// TIA Portal V15.1 export
// export: Created 2024-05-17T05:38:54.0662979Z, ExportSetting WithDefaults, DisplayName Totally Integrated Automation Portal, DisplayVersion V15.1 Update 5, DisplayName TIA Portal Openness, DisplayVersion V15.1 Update 5, DisplayName SINAMICS Startdrive Advanced, DisplayVersion V15.1, DisplayName G130, G150, S120, S150, SINAMICS MV, S210, DisplayVersion V15.1, DisplayName G110M, G120, G120C, G120D, G120P, DisplayVersion V15.1, DisplayName STEP 7 Professional, DisplayVersion V15.1 Update 5, DisplayName STEP 7 Safety, DisplayVersion V15.1, DisplayName WinCC Professional, DisplayVersion V15.1 Update 5, DisplayName SIMATIC Visualization Architect, DisplayVersion V15.1
FUNCTION_BLOCK "LVIDSTrack"   // FB1205, FBD
TITLE = LVIDS Tracking
{ S7_Optimized_Access := 'TRUE' }
VERSION : 0.1
// stored: AutoNumber false, IsIECCheckEnabled false, IsRetainMemResEnabled false, MemoryReserve 100, SetENOAutomatically False, UDAEnableTagReadback false
   VAR_INPUT
      I_DataModeManEn { ExternalAccessible := 'False'; ExternalVisible := 'False'; ExternalWritable := 'False'} : Bool;   // Data mode manual enabled
      I_OutOfUse { ExternalAccessible := 'False'; ExternalVisible := 'False'; ExternalWritable := 'False'} : Bool;   // Out of use
      I_TagID { ExternalAccessible := 'False'; ExternalVisible := 'False'; ExternalWritable := 'False'} : DInt;   // Tag identification for tracking
      I_BodyID { ExternalAccessible := 'False'; ExternalVisible := 'False'; ExternalWritable := 'False'} : DInt;   // Body identification for tracking
      I_CarrierID { ExternalAccessible := 'False'; ExternalVisible := 'False'; ExternalWritable := 'False'} : DInt;   // Carrier identification for tracking
      I_MixNbr { ExternalAccessible := 'False'; ExternalVisible := 'False'; ExternalWritable := 'False'} : DInt;   // Mixnumber for tracking
      I_BodyType1 { ExternalAccessible := 'False'; ExternalVisible := 'False'; ExternalWritable := 'False'} : DInt;   // Bodytype1 for tracking
      I_PopID { ExternalAccessible := 'False'; ExternalVisible := 'False'; ExternalWritable := 'False'} : UDInt;   // Spare Data / PopID
      I_PopIDSuffix { ExternalAccessible := 'False'; ExternalVisible := 'False'; ExternalWritable := 'False'} : Char;   // PopID suffix
      I_PopType { ExternalAccessible := 'False'; ExternalVisible := 'False'; ExternalWritable := 'False'} : UDInt;   // Pop identifier
      I_Start { ExternalAccessible := 'False'; ExternalVisible := 'False'; ExternalWritable := 'False'} : Bool;   // Start function / Start track
   END_VAR
   VAR_OUTPUT
      O_Ok { ExternalAccessible := 'False'; ExternalVisible := 'False'; ExternalWritable := 'False'} : Bool;   // Function finished / OK
      O_Nok { ExternalAccessible := 'False'; ExternalVisible := 'False'; ExternalWritable := 'False'} : Bool;   // NOK
      O_Busy { ExternalAccessible := 'False'; ExternalVisible := 'False'; ExternalWritable := 'False'} : Bool;   // Busy
      O_Status { ExternalAccessible := 'False'; ExternalVisible := 'False'; ExternalWritable := 'False'} : Int;   // Status ( < 0 : Fault ; 0 : No status; 1 : Success ; > 1 : Busy)
      O_Alarm { ExternalAccessible := 'False'; ExternalVisible := 'False'; ExternalWritable := 'False'} : Bool;   // Alarm
   END_VAR
   VAR_IN_OUT
      IO_VIDS : "VIDS";   // VIDS - internal record
      IO_Alarm : "Alarm";   // Alarm
      H_Track : "H_LVIDSTrack";   // Animation
      H_HMI : "H_HMI";   // Animation
   END_VAR
   VAR
      BtnManTrack { ExternalAccessible := 'False'; ExternalVisible := 'False'; ExternalWritable := 'False'} : Bool;
      BtnManForce { ExternalAccessible := 'False'; ExternalVisible := 'False'; ExternalWritable := 'False'} : Bool;
      BtnManOK { ExternalAccessible := 'False'; ExternalVisible := 'False'; ExternalWritable := 'False'} : Bool;
      BlockAutoStart { ExternalAccessible := 'False'; ExternalVisible := 'False'; ExternalWritable := 'False'} : Bool;
      RSAutoBlock { ExternalAccessible := 'False'; ExternalVisible := 'False'; ExternalWritable := 'False'} : Bool;
      TagIDMem { ExternalAccessible := 'False'; ExternalVisible := 'False'; ExternalWritable := 'False'} : DWord;
      BodyNbrMem { ExternalAccessible := 'False'; ExternalVisible := 'False'; ExternalWritable := 'False'} : DWord;
      MixNbrMem { ExternalAccessible := 'False'; ExternalVisible := 'False'; ExternalWritable := 'False'} : DWord;
      CarrierIDMem { ExternalAccessible := 'False'; ExternalVisible := 'False'; ExternalWritable := 'False'} : DWord;
      BodyType1Mem { ExternalAccessible := 'False'; ExternalVisible := 'False'; ExternalWritable := 'False'} : DWord;
      PopIDMem { ExternalAccessible := 'False'; ExternalVisible := 'False'; ExternalWritable := 'False'} : DWord;
      PopIDSuffixMem { ExternalAccessible := 'False'; ExternalVisible := 'False'; ExternalWritable := 'False'} : Char;
      PopTypeMem { ExternalAccessible := 'False'; ExternalVisible := 'False'; ExternalWritable := 'False'} : DWord;
      StartEdg { ExternalAccessible := 'False'; ExternalVisible := 'False'; ExternalWritable := 'False'} : Bool;   // Edge of start tracking
      StartPls { ExternalAccessible := 'False'; ExternalVisible := 'False'; ExternalWritable := 'False'} : Bool;
      StartTrackEdge2 { ExternalAccessible := 'False'; ExternalVisible := 'False'; ExternalWritable := 'False'} : Bool;   // Edge of start tracking
      StartCmdMem { ExternalAccessible := 'False'; ExternalVisible := 'False'; ExternalWritable := 'False'} : Bool;   // Memory of start command
      FinishPls { ExternalAccessible := 'False'; ExternalVisible := 'False'; ExternalWritable := 'False'} : Bool;   // Pulse of finish tracking
      FinishEdge { ExternalAccessible := 'False'; ExternalVisible := 'False'; ExternalWritable := 'False'} : Bool;   // Edge of finish tracking
      Status { ExternalAccessible := 'False'; ExternalVisible := 'False'; ExternalWritable := 'False'} : Int;   // Status
      Alarm { ExternalAccessible := 'False'; ExternalVisible := 'False'; ExternalWritable := 'False'} : Bool;
      Ok { ExternalAccessible := 'False'; ExternalVisible := 'False'; ExternalWritable := 'False'} : Bool;
      Nok { ExternalAccessible := 'False'; ExternalVisible := 'False'; ExternalWritable := 'False'} : Bool;
      BtnManConfirmVisible { ExternalAccessible := 'False'; ExternalVisible := 'False'; ExternalWritable := 'False'} : Word;
      BtnManConfirmGreen { ExternalAccessible := 'False'; ExternalVisible := 'False'; ExternalWritable := 'False'} : Word;
      BtnManForceVisible { ExternalAccessible := 'False'; ExternalVisible := 'False'; ExternalWritable := 'False'} : Word;
      BtnManForceGreen { ExternalAccessible := 'False'; ExternalVisible := 'False'; ExternalWritable := 'False'} : Word;
   END_VAR
   VAR_TEMP
      TempNotUsedBool : Bool;
   END_VAR
   VAR CONSTANT
      CMD_TRACK : DWord := 4001;
      OFF : Word := 2#0000000000000000;
      ENABLE : Word := 2#0000000000000001;
      VISIBLE : Word := 2#0000000000000010;
      COLOUR_GREY : Word := 2#0000000000010000;
      COLOUR_WHITE : Word := 2#0000000000100000;
      COLOUR_GREEN : Word := 2#0000000001000000;
      COLOUR_RED : Word := 2#0000000010000000;
      COLOUR_BLUE_FLASH : Word := 2#0000000100000000;
   END_VAR
   VAR_TEMP   // added for the SCL form of the ladder/FBD networks
      _w1 : Bool;
   END_VAR
BEGIN

REGION Network 1: **** 4.4 - Machine status - Input from HMI - Buttons
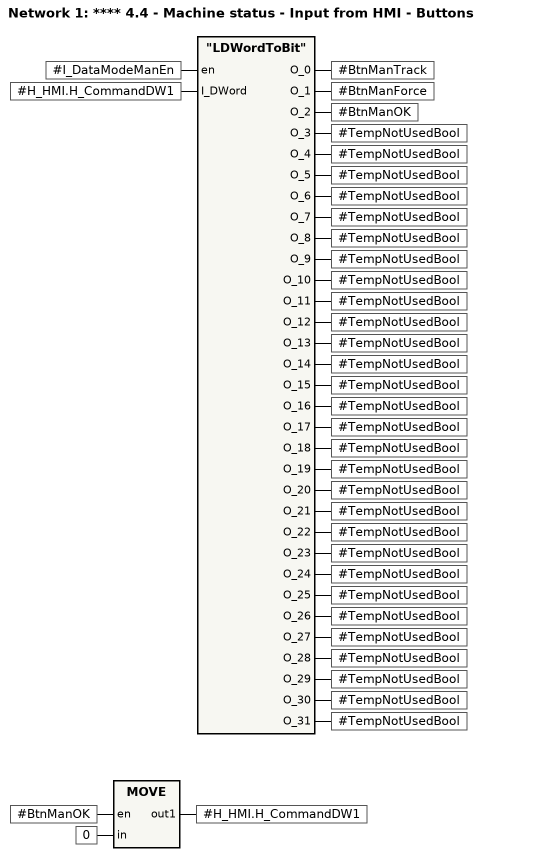
   IF #I_DataModeManEn THEN
       "LDWordToBit"(I_DWord := #H_HMI.H_CommandDW1,
                     O_0 => #BtnManTrack,
                     O_1 => #BtnManForce,
                     O_2 => #BtnManOK,
                     O_3 => #TempNotUsedBool,
                     O_4 => #TempNotUsedBool,
                     O_5 => #TempNotUsedBool,
                     O_6 => #TempNotUsedBool,
                     O_7 => #TempNotUsedBool,
                     O_8 => #TempNotUsedBool,
                     O_9 => #TempNotUsedBool,
                     O_10 => #TempNotUsedBool,
                     O_11 => #TempNotUsedBool,
                     O_12 => #TempNotUsedBool,
                     O_13 => #TempNotUsedBool,
                     O_14 => #TempNotUsedBool,
                     O_15 => #TempNotUsedBool,
                     O_16 => #TempNotUsedBool,
                     O_17 => #TempNotUsedBool,
                     O_18 => #TempNotUsedBool,
                     O_19 => #TempNotUsedBool,
                     O_20 => #TempNotUsedBool,
                     O_21 => #TempNotUsedBool,
                     O_22 => #TempNotUsedBool,
                     O_23 => #TempNotUsedBool,
                     O_24 => #TempNotUsedBool,
                     O_25 => #TempNotUsedBool,
                     O_26 => #TempNotUsedBool,
                     O_27 => #TempNotUsedBool,
                     O_28 => #TempNotUsedBool,
                     O_29 => #TempNotUsedBool,
                     O_30 => #TempNotUsedBool,
                     O_31 => #TempNotUsedBool);
   END_IF;
   IF #BtnManOK THEN #H_HMI.H_CommandDW1 := 0; END_IF;
END_REGION

REGION Network 2: *** 4.4 - Machine status - Calculated *** / **** 4.4 - Machine status - Calculated *** Begin request
   // Start request memory
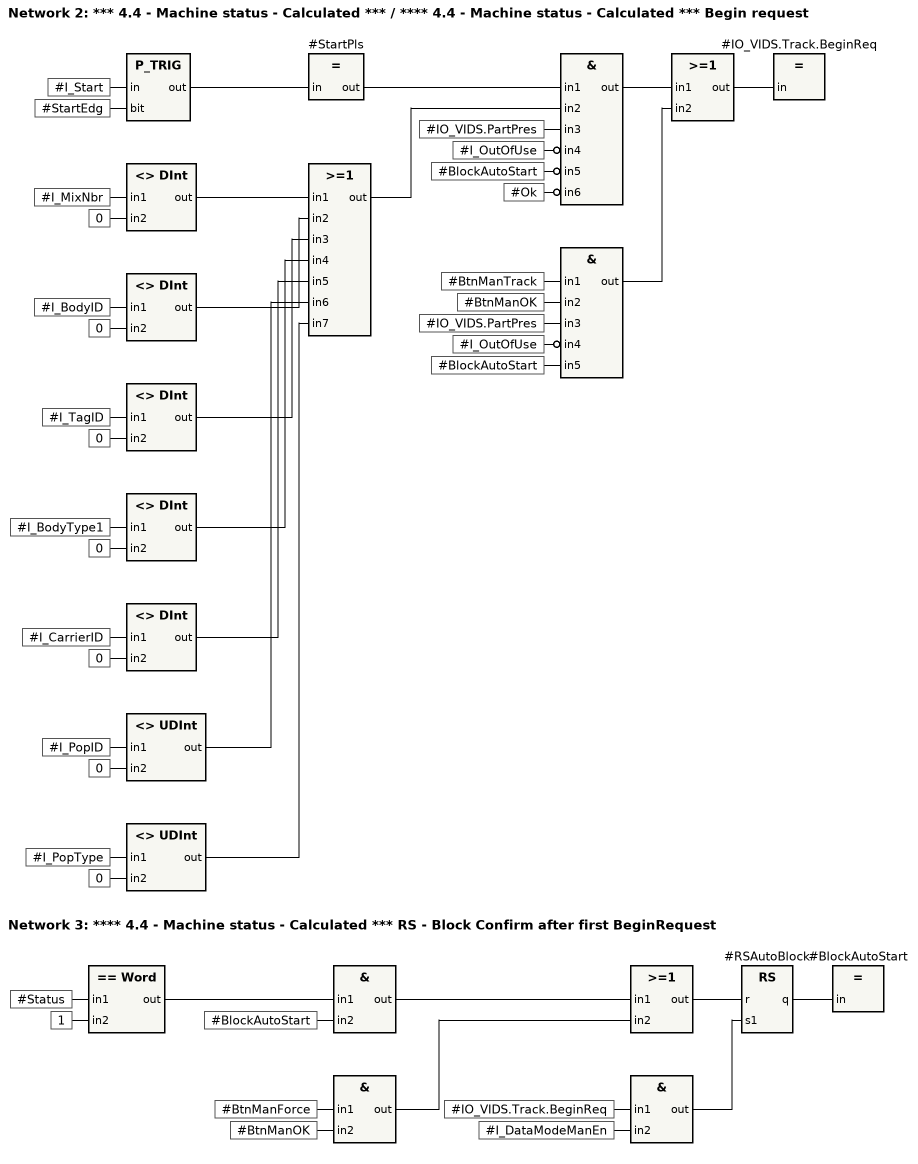
   #_w1 := #I_Start AND NOT #StartEdg;   // rising edge
   #StartEdg := #I_Start;
   #StartPls := #_w1;
   #IO_VIDS.Track.BeginReq := (#_w1 AND ((#I_MixNbr <> 0) OR (#I_BodyID <> 0) OR (#I_TagID <> 0) OR (#I_BodyType1 <> 0) OR (#I_CarrierID <> 0) OR (#I_PopID <> 0) OR (#I_PopType <> 0)) AND #IO_VIDS.PartPres AND NOT #I_OutOfUse AND NOT #BlockAutoStart AND NOT #Ok) OR (#BtnManTrack AND #BtnManOK AND #IO_VIDS.PartPres AND NOT #I_OutOfUse AND #BlockAutoStart);
END_REGION

REGION Network 3: **** 4.4 - Machine status - Calculated *** RS - Block Confirm after first BeginRequest
   IF ((#Status = 1) AND #BlockAutoStart) OR (#BtnManForce AND #BtnManOK) THEN
       #RSAutoBlock := FALSE;   // RS flip-flop
   END_IF;
   IF #IO_VIDS.Track.BeginReq AND #I_DataModeManEn THEN #RSAutoBlock := TRUE; END_IF;
   #BlockAutoStart := #RSAutoBlock;
END_REGION

REGION Network 4: **** 4.4 - Machine status - Calculated *** Memorize parameters
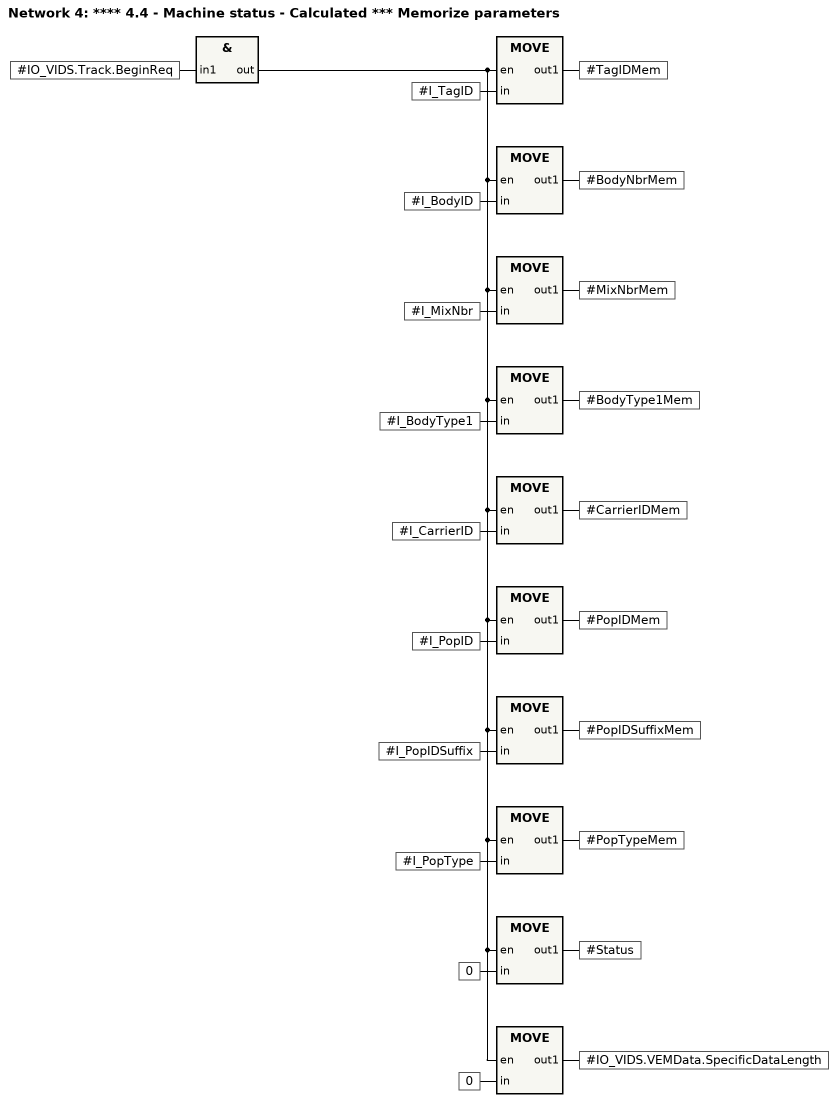
   IF #IO_VIDS.Track.BeginReq THEN
       #TagIDMem := #I_TagID;
       #BodyNbrMem := #I_BodyID;
       #MixNbrMem := #I_MixNbr;
       #BodyType1Mem := #I_BodyType1;
       #CarrierIDMem := #I_CarrierID;
       #PopIDMem := #I_PopID;
       #PopIDSuffixMem := #I_PopIDSuffix;
       #PopTypeMem := #I_PopType;
       #Status := 0;
       #IO_VIDS.VEMData.SpecificDataLength := 0;
   END_IF;
END_REGION

REGION Network 5: *** 4.4 - Machine status - Calculated *** / **** 4.4 - Machine status - Calculated *** Ok to begin
   // Data mode auto - Begin pulse
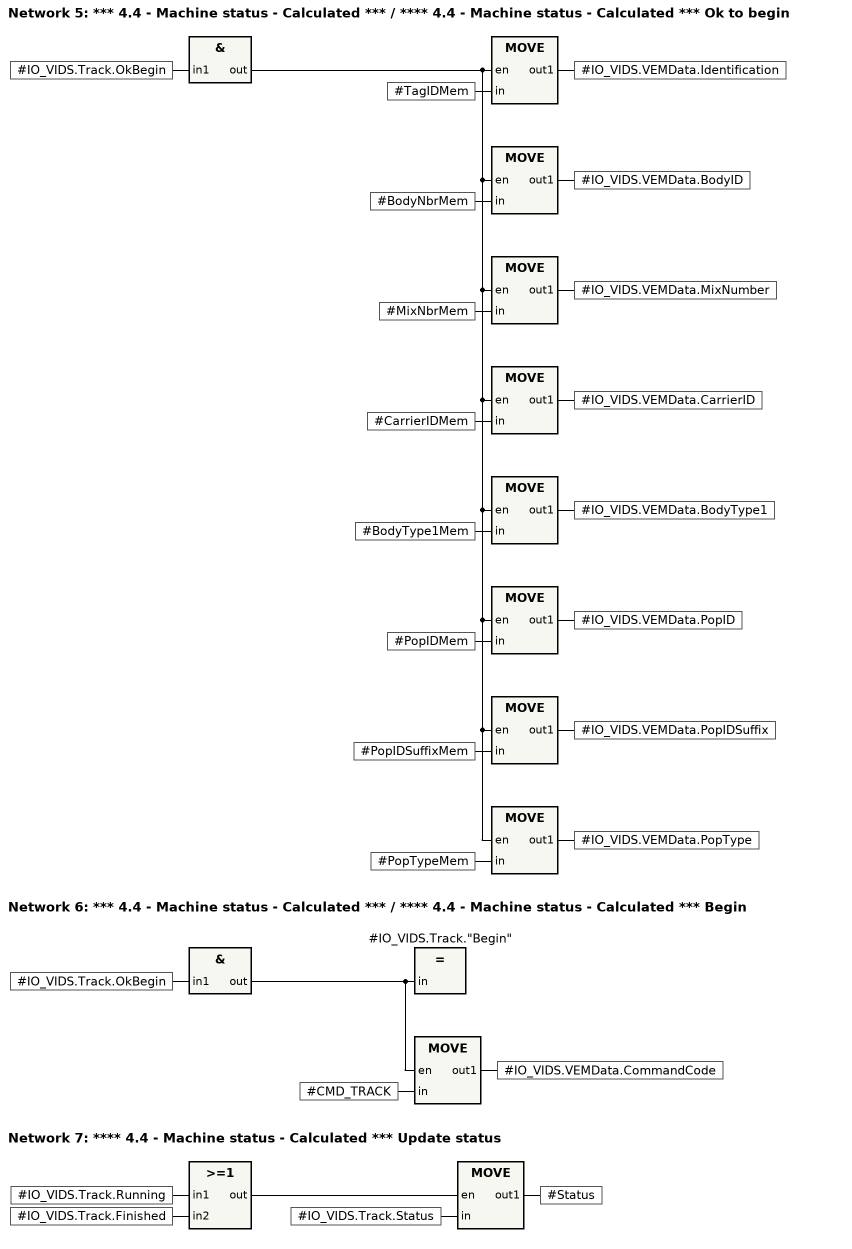
   IF #IO_VIDS.Track.OkBegin THEN
       #IO_VIDS.VEMData.Identification := #TagIDMem;
       #IO_VIDS.VEMData.BodyID := #BodyNbrMem;
       #IO_VIDS.VEMData.MixNumber := #MixNbrMem;
       #IO_VIDS.VEMData.CarrierID := #CarrierIDMem;
       #IO_VIDS.VEMData.BodyType1 := #BodyType1Mem;
       #IO_VIDS.VEMData.PopID := #PopIDMem;
       #IO_VIDS.VEMData.PopIDSuffix := #PopIDSuffixMem;
       #IO_VIDS.VEMData.PopType := #PopTypeMem;
   END_IF;
END_REGION

REGION Network 6: *** 4.4 - Machine status - Calculated *** / **** 4.4 - Machine status - Calculated *** Begin
   // Data mode auto - Begin pulse
   #IO_VIDS.Track."Begin" := #IO_VIDS.Track.OkBegin;
   IF #IO_VIDS.Track.OkBegin THEN #IO_VIDS.VEMData.CommandCode := #CMD_TRACK; END_IF;
END_REGION

REGION Network 7: **** 4.4 - Machine status - Calculated *** Update status
   IF #IO_VIDS.Track.Running OR #IO_VIDS.Track.Finished THEN #Status := #IO_VIDS.Track.Status; END_IF;
END_REGION

REGION Network 8: *** 8 - Outputs *** / **** 4.4 - Machine status - Calculated *** Finished, OK
   // Feedback to process - Tracking finished
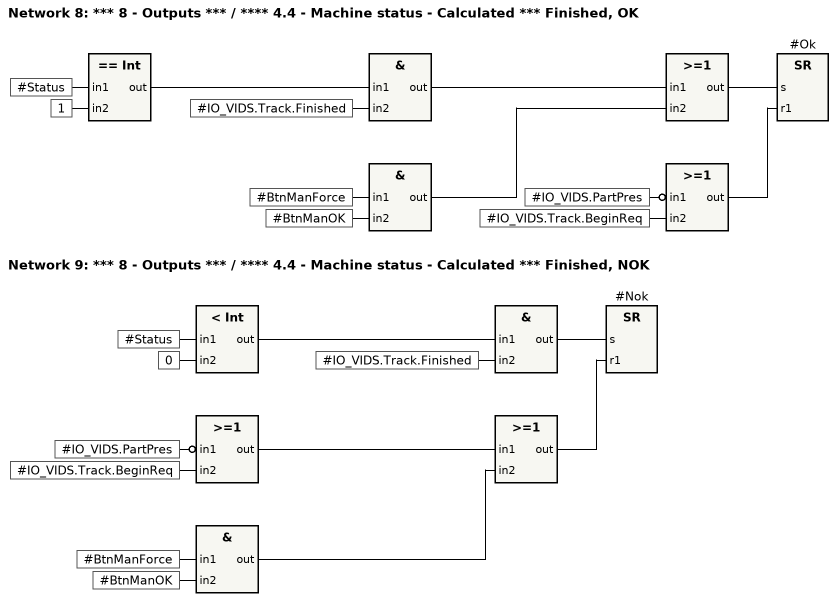
   IF ((#Status = 1) AND #IO_VIDS.Track.Finished) OR (#BtnManForce AND #BtnManOK) THEN
       #Ok := TRUE;   // SR flip-flop
   END_IF;
   IF NOT #IO_VIDS.PartPres OR #IO_VIDS.Track.BeginReq THEN #Ok := FALSE; END_IF;
END_REGION

REGION Network 9: *** 8 - Outputs *** / **** 4.4 - Machine status - Calculated *** Finished, NOK
   // Feedback to process - Tracking finished
   IF (#Status < 0) AND #IO_VIDS.Track.Finished THEN
       #Nok := TRUE;   // SR flip-flop
   END_IF;
   IF NOT #IO_VIDS.PartPres OR #IO_VIDS.Track.BeginReq OR (#BtnManForce AND #BtnManOK) THEN
       #Nok := FALSE;
   END_IF;
END_REGION

REGION Network 10: **** 4.6 - Machine status - Indication *** To HMI - Reset HMI parameters
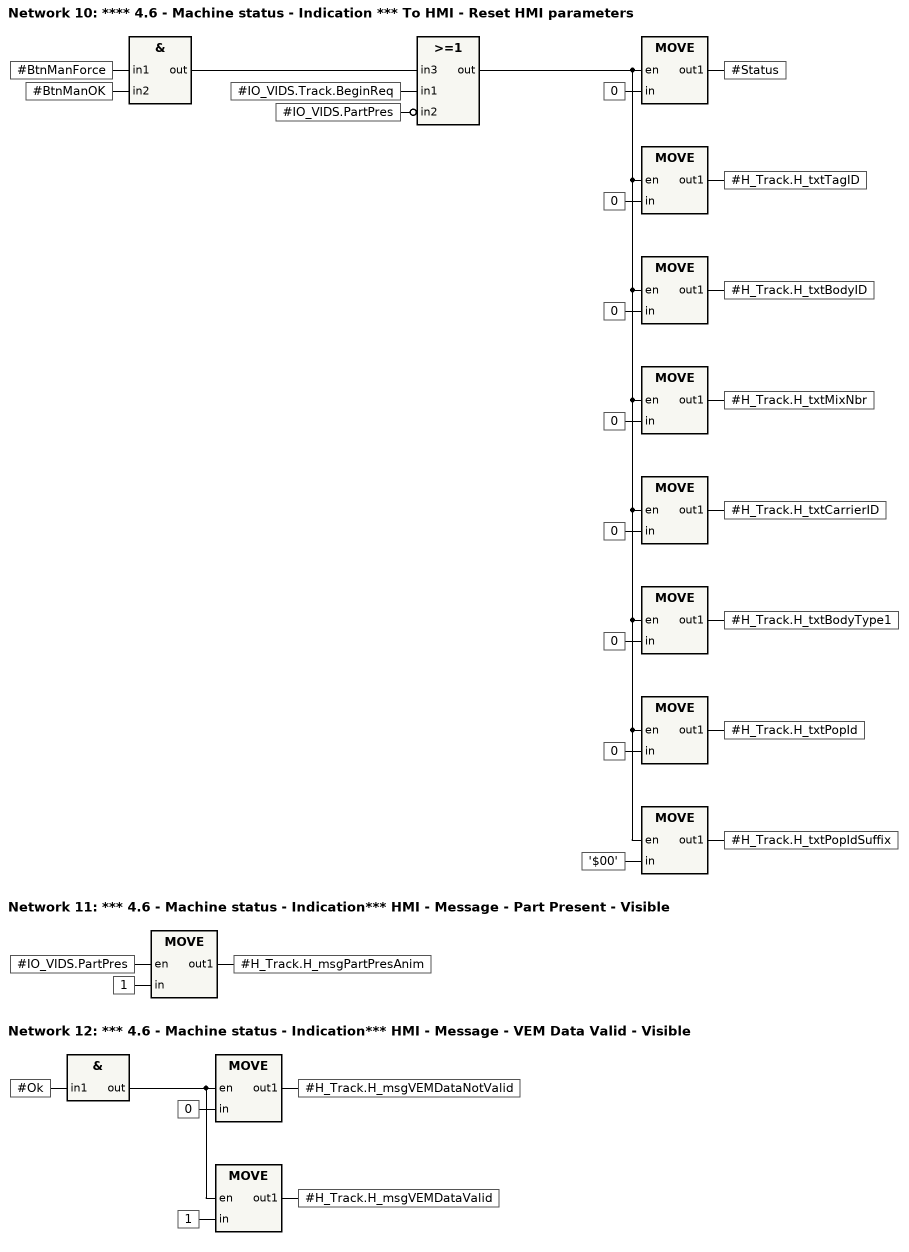
   IF (#BtnManForce AND #BtnManOK) OR #IO_VIDS.Track.BeginReq OR NOT #IO_VIDS.PartPres THEN
       #Status := 0;
       #H_Track.H_txtTagID := 0;
       #H_Track.H_txtBodyID := 0;
       #H_Track.H_txtMixNbr := 0;
       #H_Track.H_txtCarrierID := 0;
       #H_Track.H_txtBodyType1 := 0;
       #H_Track.H_txtPopId := 0;
       #H_Track.H_txtPopIdSuffix := '$00';
   END_IF;
END_REGION

REGION Network 11: *** 4.6 - Machine status - Indication*** HMI - Message - Part Present - Visible
   IF #IO_VIDS.PartPres THEN #H_Track.H_msgPartPresAnim := 1; END_IF;
END_REGION

REGION Network 12: *** 4.6 - Machine status - Indication*** HMI - Message - VEM Data Valid - Visible
   IF #Ok THEN
       #H_Track.H_msgVEMDataNotValid := 0;
       #H_Track.H_msgVEMDataValid := 1;
   END_IF;
END_REGION

REGION Network 13: *** 4.6 - Machine status - Indication*** HMI - Message - VEM Data Not Valid - Visible
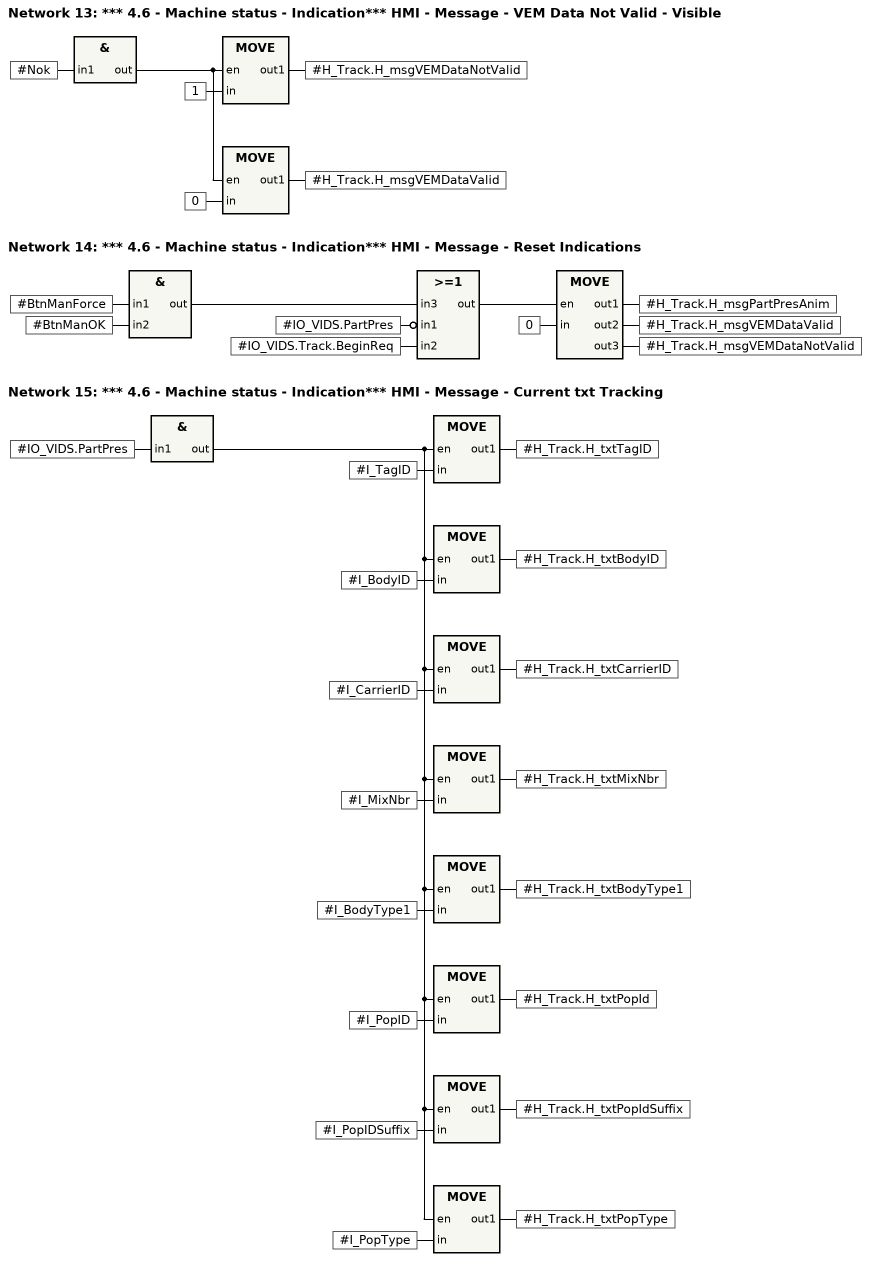
   IF #Nok THEN
       #H_Track.H_msgVEMDataNotValid := 1;
       #H_Track.H_msgVEMDataValid := 0;
   END_IF;
END_REGION

REGION Network 14: *** 4.6 - Machine status - Indication*** HMI - Message - Reset Indications
   IF (#BtnManForce AND #BtnManOK) OR NOT #IO_VIDS.PartPres OR #IO_VIDS.Track.BeginReq THEN
       #H_Track.H_msgPartPresAnim := 0;
       #H_Track.H_msgVEMDataValid := 0;
       #H_Track.H_msgVEMDataNotValid := 0;
   END_IF;
END_REGION

REGION Network 15: *** 4.6 - Machine status - Indication*** HMI - Message - Current txt Tracking
   IF #IO_VIDS.PartPres THEN
       #H_Track.H_txtTagID := #I_TagID;
       #H_Track.H_txtBodyID := #I_BodyID;
       #H_Track.H_txtCarrierID := #I_CarrierID;
       #H_Track.H_txtMixNbr := #I_MixNbr;
       #H_Track.H_txtBodyType1 := #I_BodyType1;
       #H_Track.H_txtPopId := #I_PopID;
       #H_Track.H_txtPopIdSuffix := #I_PopIDSuffix;
       #H_Track.H_txtPopType := #I_PopType;
   END_IF;
END_REGION

REGION Network 16: *** 4.6 - Machine status - Indication*** HMI - Message - Current txt Tracking Reset
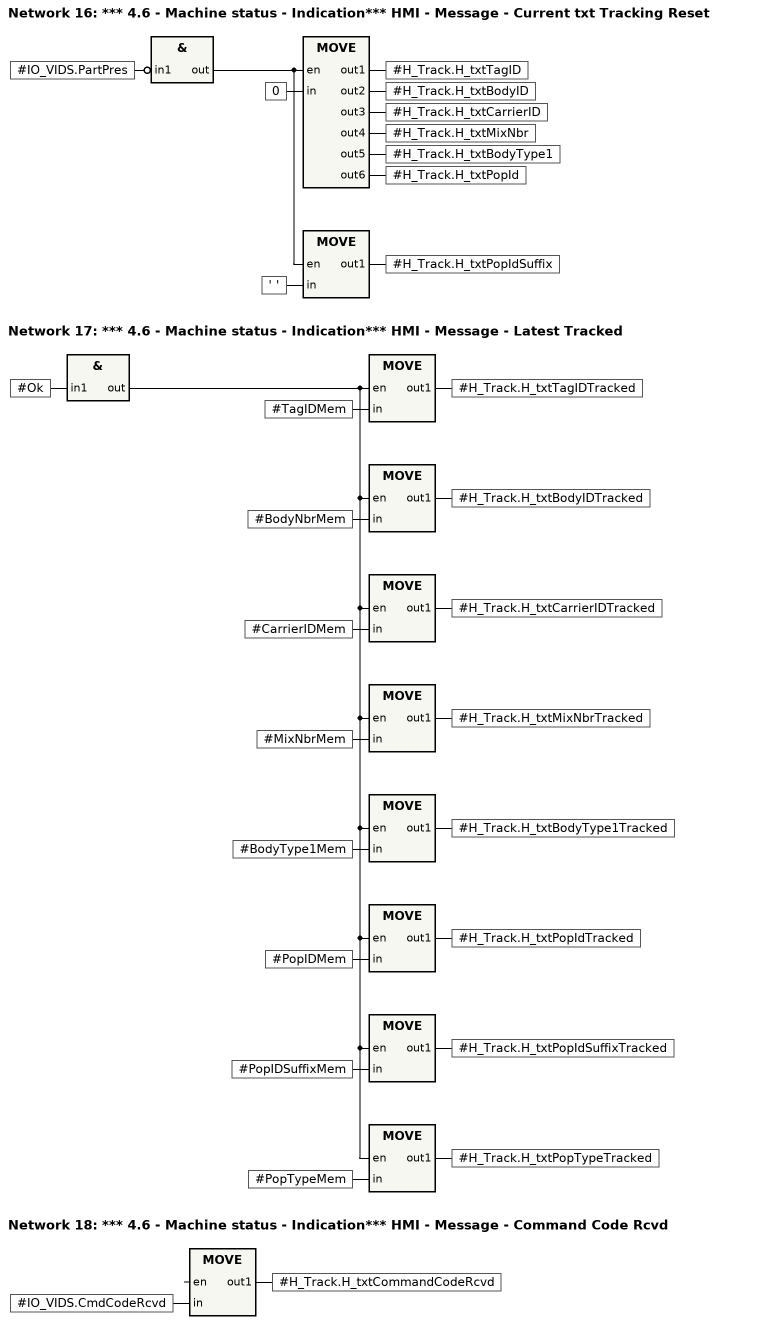
   IF NOT #IO_VIDS.PartPres THEN
       #H_Track.H_txtTagID := 0;
       #H_Track.H_txtBodyID := 0;
       #H_Track.H_txtCarrierID := 0;
       #H_Track.H_txtMixNbr := 0;
       #H_Track.H_txtBodyType1 := 0;
       #H_Track.H_txtPopId := 0;
       #H_Track.H_txtPopIdSuffix := ' ';
   END_IF;
END_REGION

REGION Network 17: *** 4.6 - Machine status - Indication*** HMI - Message - Latest Tracked
   IF #Ok THEN
       #H_Track.H_txtTagIDTracked := #TagIDMem;
       #H_Track.H_txtBodyIDTracked := #BodyNbrMem;
       #H_Track.H_txtCarrierIDTracked := #CarrierIDMem;
       #H_Track.H_txtMixNbrTracked := #MixNbrMem;
       #H_Track.H_txtBodyType1Tracked := #BodyType1Mem;
       #H_Track.H_txtPopIdTracked := #PopIDMem;
       #H_Track.H_txtPopIdSuffixTracked := #PopIDSuffixMem;
       #H_Track.H_txtPopTypeTracked := #PopTypeMem;
   END_IF;
END_REGION

REGION Network 18: *** 4.6 - Machine status - Indication*** HMI - Message - Command Code Rcvd
   #H_Track.H_txtCommandCodeRcvd := #IO_VIDS.CmdCodeRcvd;
END_REGION

REGION Network 19: *** 4.6 - Machine status - Indication*** HMI - Message - Command Code Sent
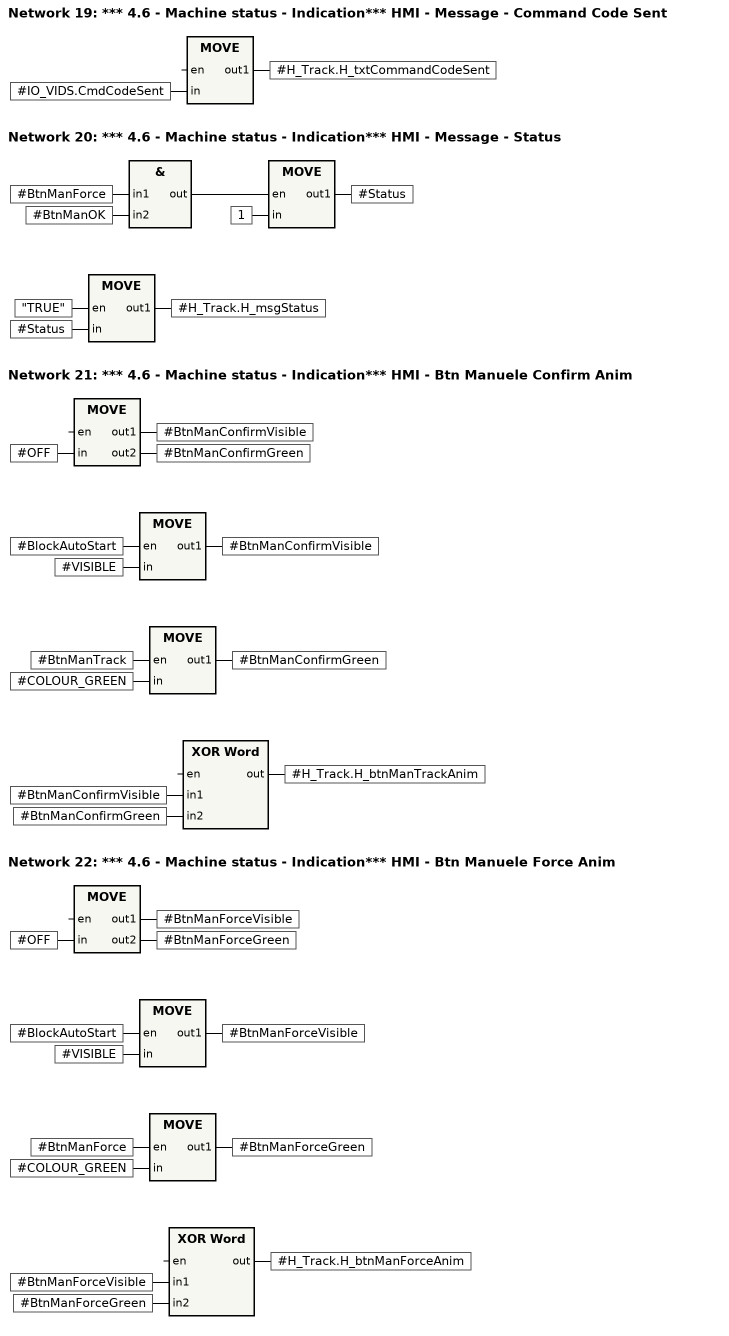
   #H_Track.H_txtCommandCodeSent := #IO_VIDS.CmdCodeSent;
END_REGION

REGION Network 20: *** 4.6 - Machine status - Indication*** HMI - Message - Status
   IF #BtnManForce AND #BtnManOK THEN #Status := 1; END_IF;
   IF "TRUE" THEN #H_Track.H_msgStatus := #Status; END_IF;
END_REGION

REGION Network 21: *** 4.6 - Machine status - Indication*** HMI - Btn Manuele Confirm Anim
   #BtnManConfirmVisible := #OFF;
   #BtnManConfirmGreen := #OFF;
   IF #BlockAutoStart THEN #BtnManConfirmVisible := #VISIBLE; END_IF;
   IF #BtnManTrack THEN #BtnManConfirmGreen := #COLOUR_GREEN; END_IF;
   #H_Track.H_btnManTrackAnim := #BtnManConfirmVisible XOR #BtnManConfirmGreen;
END_REGION

REGION Network 22: *** 4.6 - Machine status - Indication*** HMI - Btn Manuele Force Anim
   #BtnManForceVisible := #OFF;
   #BtnManForceGreen := #OFF;
   IF #BlockAutoStart THEN #BtnManForceVisible := #VISIBLE; END_IF;
   IF #BtnManForce THEN #BtnManForceGreen := #COLOUR_GREEN; END_IF;
   #H_Track.H_btnManForceAnim := #BtnManForceVisible XOR #BtnManForceGreen;
END_REGION

REGION Network 23: *** 4.6 - Machine status - Indication*** HMI - Btn Manuele Confirm Anim
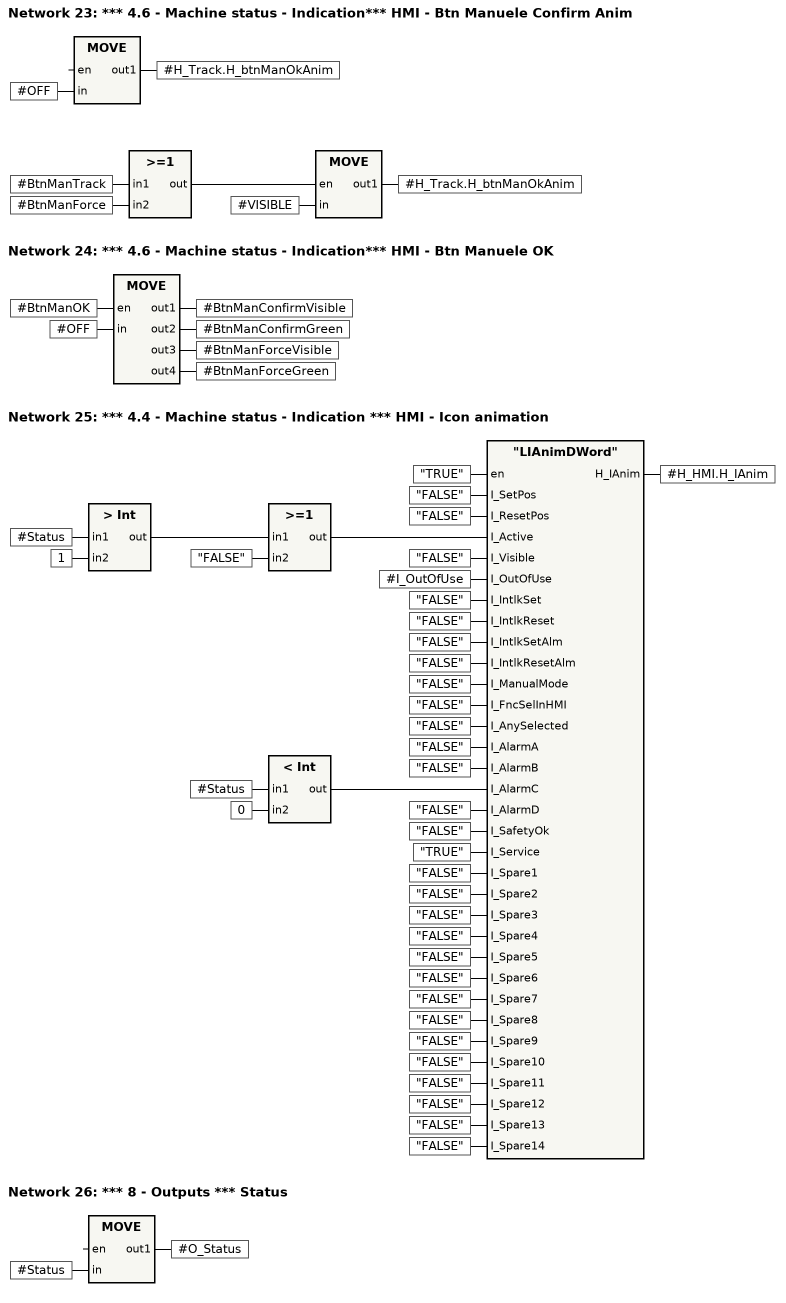
   #H_Track.H_btnManOkAnim := #OFF;
   IF #BtnManTrack OR #BtnManForce THEN #H_Track.H_btnManOkAnim := #VISIBLE; END_IF;
END_REGION

REGION Network 24: *** 4.6 - Machine status - Indication*** HMI - Btn Manuele OK
   IF #BtnManOK THEN
       #BtnManConfirmVisible := #OFF;
       #BtnManConfirmGreen := #OFF;
       #BtnManForceVisible := #OFF;
       #BtnManForceGreen := #OFF;
   END_IF;
END_REGION

REGION Network 25: *** 4.4 - Machine status - Indication *** HMI - Icon animation
   IF "TRUE" THEN
       "LIAnimDWord"(I_SetPos := "FALSE",
                     I_ResetPos := "FALSE",
                     I_Active := (#Status > 1) OR "FALSE",
                     I_Visible := "FALSE",
                     I_OutOfUse := #I_OutOfUse,
                     I_IntlkSet := "FALSE",
                     I_IntlkReset := "FALSE",
                     I_IntlkSetAlm := "FALSE",
                     I_IntlkResetAlm := "FALSE",
                     I_ManualMode := "FALSE",
                     I_FncSelInHMI := "FALSE",
                     I_AnySelected := "FALSE",
                     I_AlarmA := "FALSE",
                     I_AlarmB := "FALSE",
                     I_AlarmC := #Status < 0,
                     I_AlarmD := "FALSE",
                     I_SafetyOk := "FALSE",
                     I_Service := "TRUE",
                     I_Spare1 := "FALSE",
                     I_Spare2 := "FALSE",
                     I_Spare3 := "FALSE",
                     I_Spare4 := "FALSE",
                     I_Spare5 := "FALSE",
                     I_Spare6 := "FALSE",
                     I_Spare7 := "FALSE",
                     I_Spare8 := "FALSE",
                     I_Spare9 := "FALSE",
                     I_Spare10 := "FALSE",
                     I_Spare11 := "FALSE",
                     I_Spare12 := "FALSE",
                     I_Spare13 := "FALSE",
                     I_Spare14 := "FALSE",
                     H_IAnim => #H_HMI.H_IAnim);
   END_IF;
END_REGION

REGION Network 26: *** 8 - Outputs *** Status
   #O_Status := #Status;
END_REGION

REGION Network 27: *** 8 - Outputs *** Busy
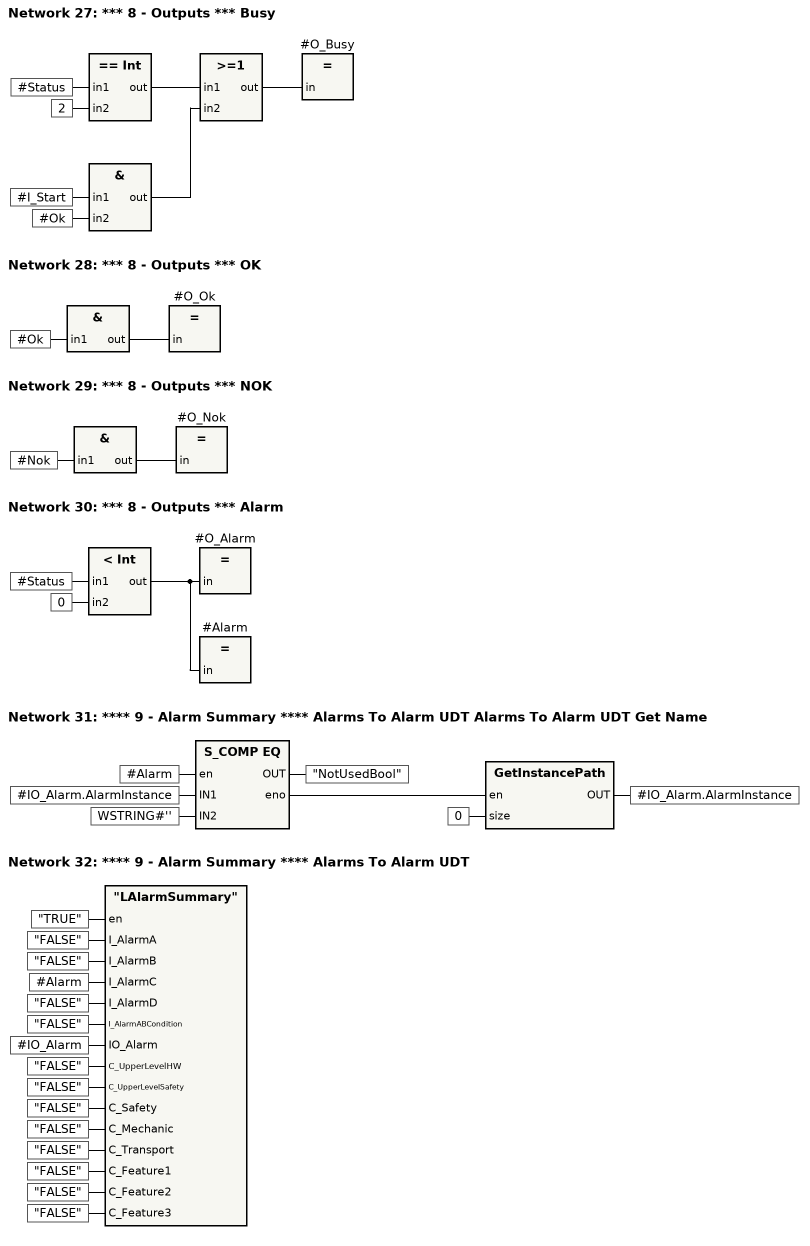
   #O_Busy := (#Status = 2) OR (#I_Start AND #Ok);
END_REGION

REGION Network 28: *** 8 - Outputs *** OK
   #O_Ok := #Ok;
END_REGION

REGION Network 29: *** 8 - Outputs *** NOK
   #O_Nok := #Nok;
END_REGION

REGION Network 30: *** 8 - Outputs *** Alarm
   #O_Alarm := #Status < 0;
   #Alarm := #O_Alarm;
END_REGION

REGION Network 31: **** 9 - Alarm Summary **** Alarms To Alarm UDT Alarms To Alarm UDT Get Name
   // Alarm / Alarm D
   S_COMP(EN := #Alarm, IN1 := #IO_Alarm.AlarmInstance, IN2 := WSTRING#'', OUT => "NotUsedBool", ENO => #_w1);
   IF #_w1 THEN GetInstancePath(size := 0, OUT => #IO_Alarm.AlarmInstance); END_IF;
END_REGION

REGION Network 32: **** 9 - Alarm Summary **** Alarms To Alarm UDT
   // Alarm / Alarm D
   IF "TRUE" THEN
       "LAlarmSummary"(I_AlarmA := "FALSE",
                       I_AlarmB := "FALSE",
                       I_AlarmC := #Alarm,
                       I_AlarmD := "FALSE",
                       I_AlarmABCondition := "FALSE",
                       IO_Alarm := #IO_Alarm,
                       C_UpperLevelHW := "FALSE",
                       C_UpperLevelSafety := "FALSE",
                       C_Safety := "FALSE",
                       C_Mechanic := "FALSE",
                       C_Transport := "FALSE",
                       C_Feature1 := "FALSE",
                       C_Feature2 := "FALSE",
                       C_Feature3 := "FALSE");
   END_IF;
END_REGION
END_FUNCTION_BLOCK
